// TIA Portal V20 export
VAR_GLOBAL   // PLC tag table "Safety"
END_VAR
